FUNCTION_BLOCK FB_Roboterachsensteuerung
VAR_INPUT
	// Steuereingang
	bEnable : BOOL;
	bExecute : BOOL;
	rPosition : REAL;
	bRefSens: BOOL;
END_VAR
VAR_OUTPUT
	eState : eBetriebszustand;
END_VAR
VAR
	nState : INT := 0;
	rVelocity : REAL;
	rAccelaration : REAL;
	
	// Motion Blöcke Tc2_Mc2
	mcReset : MC_Reset;
	mcPower : MC_Power;
	mcAbsolute : MC_MoveAbsolute;
	mcHome : MC_Home;
	
END_VAR
VAR_IN_OUT
	ax : AXIS_REF;
END_VAR

ax.ReadStatus();

mcPower(
	Axis:= ax, 
	Enable:= bEnable, 
	Enable_Positive:= TRUE, 
	Enable_Negative:= TRUE, 
	Override:= , 
	BufferMode:= , 
	Options:= , 
	Status=> , 
	Busy=> , 
	Error=> , 
	ErrorID=> );
	
mcReset(
	Axis:= ax, 
	Execute:= , 
	Done=> , 
	Busy=> , 
	Error=> , 
	ErrorID=> );

mcAbsolute(
	Axis:= ax, 
	Execute:= , 
	Position:= , 
	Velocity:= rVelocity, 
	Acceleration:= rAccelaration, 
	Deceleration:= rAccelaration, 
	Jerk:= , 
	BufferMode:= , 
	Options:= , 
	Done=> , 
	Busy=> , 
	Active=> , 
	CommandAborted=> , 
	Error=> , 
	ErrorID=> );

mcHome(
	Axis:= ax, 
	Execute:= , 
	Position:= , 
	HomingMode:= , 
	BufferMode:= , 
	Options:= , 
	bCalibrationCam:= NOT bRefSens, 
	Done=> , 
	Busy=> , 
	Active=> , 
	CommandAborted=> , 
	Error=> , 
	ErrorID=> );
	
	

CASE nState OF
	0: // OFF
	eState := eBetriebszustand.OFF;
	mcPower.Enable := TRUE;
	mcReset.Execute := FALSE;
	
	IF bEnable THEN
		nState := 10; // INIT-Reset
	END_IF
	
	10: // INIT-Reset
	eState := eBetriebszustand.INIT;
		
	mcPower.Enable := FALSE;
	mcReset.Execute := TRUE;
	
	IF mcReset.Done THEN
		nState := 11; // INIT-Power
	END_IF
	
	11: // INIT-Power
	eState := eBetriebszustand.INIT;
		
	mcPower.Enable := TRUE;
	mcReset.Execute := FALSE;
	
	IF mcPower.Status AND NOT ax.Status.Homed THEN
		nState := 12; // INIT-Home
	ELSIF mcPower.Status AND ax.Status.Homed THEN
		nState := 20; // READY
	END_IF
	
	12: // INIT-Home
	eState := eBetriebszustand.INIT;
			
	mcHome.Execute := TRUE;
	
	IF mcHome.Done THEN
		nState := 20; // READY
	END_IF
	
	20: // READY
	eState := eBetriebszustand.READY;
			
	IF bExecute THEN
		nState := 30; // PROD-Bewegen
	END_IF
	
	30: // PROD-Bewegen
	eState := eBetriebszustand.PROD;
	METH_MoveAxis(rPosition);
	//mcAbsolute.Position := rPosition;
	mcAbsolute.Velocity := 30;
	mcAbsolute.Acceleration := 60;
	
	IF mcAbsolute.Done THEN
		nState := 40; // DONE
	END_IF
	
	40: // DONE
	eState := eBetriebszustand.DONE;
	mcAbsolute.Execute := FALSE;
	IF NOT bExecute THEN
		nState := 20; // READY
	END_IF
	
END_CASE

METHOD METH_MoveAxis : BOOL
VAR_INPUT
	rPos	: REAL;
END_VAR
mcAbsolute(
	Axis:= ax, 
	Execute:= TRUE, 
	Position:= rPos, 
	Velocity:= rVelocity, 
	Acceleration:= rAccelaration, 
	Deceleration:= rAccelaration, 
	Jerk:= , 
	BufferMode:= , 
	Options:= , 
	Done=> , 
	Busy=> , 
	Active=> , 
	CommandAborted=> , 
	Error=> , 
	ErrorID=> );
END_METHOD

END_FUNCTION_BLOCK

(* stored: Version 1.1.0.1, ProductVersion 3.1.4024.15
   POU FB_Roboterachsensteuerung: Id {0ef852b6-e5ca-4c53-bced-af77fdb653f5}, SpecialFunc None
   Method METH_MoveAxis: Id {19c464a0-8720-46f4-acb9-6acd54af2ded} *)
